// TIA Portal V16 export
// export: Created 2025-05-30T16:30:15.279761Z, ExportSetting WithDefaults, DisplayName Totally Integrated Automation Portal, DisplayVersion V16, DisplayName TIA Portal Version Control Interface, DisplayVersion V16, DisplayName TIA Portal Openness, DisplayVersion V16, DisplayName STEP 7 Professional, DisplayVersion V16, DisplayName STEP 7 Safety, DisplayVersion V16, DisplayName WinCC Advanced, DisplayVersion V16
FUNCTION "9 - OVERIG" : Void   // FC6, LAD
TITLE = Other - Testing
VERSION : 0.1
// stored: AutoNumber true, IsIECCheckEnabled false, UDAEnableTagReadback false
   VAR_TEMP
      Encoder : Int;
      Gate : Bool;
      GATESTP : Bool;
      OTERRA : Bool;
      Direct : Bool;
      Prepar : Bool;
      CMPV1 : Bool;
      CMPV2 : Bool;
      RESSYNC : Bool;
      RESZERO : Bool;
      OTERR : Bool;
   END_VAR
BEGIN

REGION Network 1: SAFETY - OVERRIDE
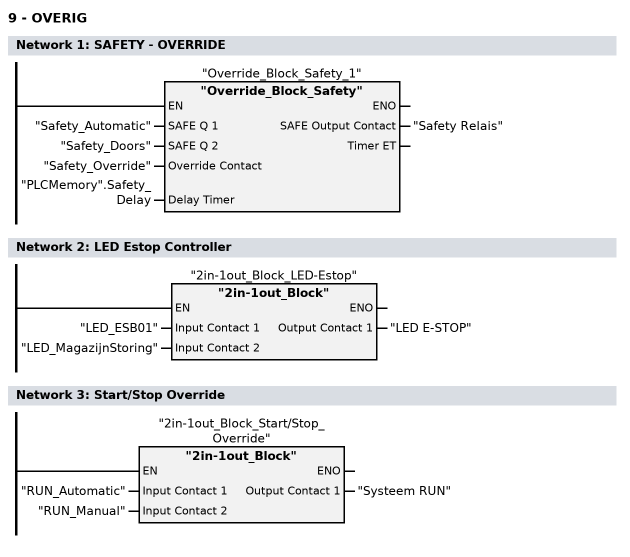
   RUNG wire#powerrail
      "Override_Block_Safety_1"("SAFE Q 1" := "Safety_Automatic", "SAFE Q 2" := "Safety_Doors", "Override Contact" := "Safety_Override", "Delay Timer" := "PLCMemory".Safety_Delay, "SAFE Output Contact" => "Safety Relais", "Timer ET" =>)
   END_RUNG
   // the same network as SCL:
   "Override_Block_Safety_1"("SAFE Q 1" := "Safety_Automatic",   // "Override_Block_Safety"
                           "SAFE Q 2" := "Safety_Doors",
                           "Override Contact" := "Safety_Override",
                           "Delay Timer" := "PLCMemory".Safety_Delay,
                           "SAFE Output Contact" => "Safety Relais");
END_REGION

REGION Network 2: LED Estop Controller
   RUNG wire#powerrail
      "2in-1out_Block_LED-Estop"("Input Contact 1" := "LED_ESB01", "Input Contact 2" := "LED_MagazijnStoring", "Output Contact 1" => "LED E-STOP")
   END_RUNG
   // the same network as SCL:
   "2in-1out_Block_LED-Estop"("Input Contact 1" := "LED_ESB01",   // "2in-1out_Block"
                           "Input Contact 2" := "LED_MagazijnStoring",
                           "Output Contact 1" => "LED E-STOP");
END_REGION

REGION Network 3: Start/Stop Override
   RUNG wire#powerrail
      "2in-1out_Block_Start/Stop_Override"("Input Contact 1" := "RUN_Automatic", "Input Contact 2" := "RUN_Manual", "Output Contact 1" => "Systeem RUN")
   END_RUNG
   // the same network as SCL:
   "2in-1out_Block_Start/Stop_Override"("Input Contact 1" := "RUN_Automatic",   // "2in-1out_Block"
                           "Input Contact 2" := "RUN_Manual",
                           "Output Contact 1" => "Systeem RUN");
END_REGION
END_FUNCTION
